FUNCTION F_Logger : STRING;
VAR_INPUT
	LogSeverity : E_LogSeverity_Ish;
	Message : T_MaxString;
END_VAR

IF ( LogSeverity < E_LogSeverity_Ish.None ) 
	AND_THEN ( LogSeverity >= LogConfig.LogLevel ) THEN
	
	ADSLOGSTR(LogSeverity OR ADSLOG_MSGTYPE_LOG, Message, '');
	F_Logger := Message;
	
END_IF

END_FUNCTION

(* stored: Version 1.1.0.1, ProductVersion 3.1.4022.18
   POU F_Logger: Id {852c98e6-427b-41a5-90fd-93ad32d4751e}, SpecialFunc None *)
